// TIA Portal V20 export
TYPE "typeSequenceControlNodeInterafceSTKJobInterface"
// stored: Namespace Unit1.Em7
   STRUCT
      commands : "Unit1.Em7.typeSequenceControlNodeInterafceSTKJobInterfaceCommands";
      monitoring { S7_SetPoint := 'True'} : "Unit1.Em7.typeSequenceControlNodeInterafceSTKJobInterfaceMonitoring";
   END_STRUCT;
END_TYPE
